FUNCTION_BLOCK FB_EventArray
VAR_INPUT
END_VAR
VAR_OUTPUT
END_VAR
VAR
END_VAR

END_FUNCTION_BLOCK

(* stored: Version 1.1.0.1, ProductVersion 3.1.4024.12
   POU FB_EventArray: Id {4c5b9bd1-4620-46c9-9b9e-0df77ea88e21}, SpecialFunc None *)
